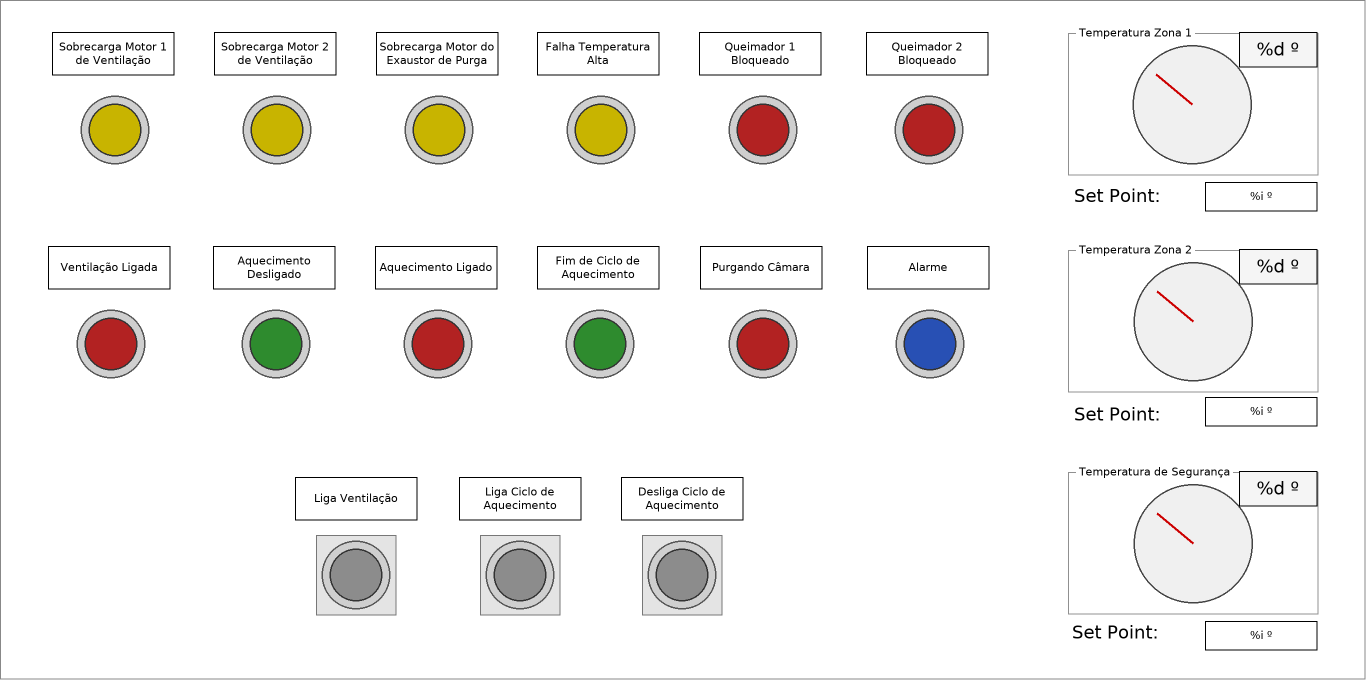
VISUALIZATION Manu021  // 1366x680
    Lamp1 (75,90 80x80), variable: GVL.sobrecarga_M1_vent_021, style: Lamp-Lamp1-Yellow
    Lamp1 (237,90 80x80), variable: GVL.sobrecarga_M2_vent_021, style: Lamp-Lamp1-Yellow
    Lamp1 (399,90 80x80), variable: GVL.sobrecarga_Purga_021, style: Lamp-Lamp1-Yellow
    Lamp1 (561,90 80x80), variable: GVL.falhaTempHigh_021, style: Lamp-Lamp1-Yellow
    Lamp1 (723,90 80x80), variable: GVL.queimador1_block_021, style: Lamp-Lamp1-Red
    Lamp1 (889,90 80x80), variable: GVL.queimador2_block_021, style: Lamp-Lamp1-Red
    Rectangle (52,32 122x43), "Sobrecarga Motor 1 de Ventilação"
    Rectangle (214,32 122x43), "Sobrecarga Motor 2 de Ventilação"
    Rectangle (376,32 122x43), "Sobrecarga Motor do Exaustor de Purga"
    Rectangle (537,32 122x43), "Falha Temperatura Alta"
    Rectangle (699,32 122x43), "Queimador 1 Bloqueado"
    Rectangle (866,32 122x43), "Queimador 2 Bloqueado"
    Lamp1 (71,304 80x80), variable: GVL.ventilacao_Ligada_021, style: Lamp-Lamp1-Red
    Rectangle (48,246 122x43), "Ventilação Ligada"
    Lamp1 (236,304 80x80), variable: GVL.aquecimento_Desligado_021, style: Lamp-Lamp1-Green
    Rectangle (213,246 122x43), "Aquecimento Desligado"
    Lamp1 (398,304 80x80), variable: GVL.aquecimento_Ligado_021, style: Lamp-Lamp1-Red
    Rectangle (375,246 122x43), "Aquecimento Ligado"
    Lamp1 (560,304 80x80), variable: GVL.fimCicloAquecimento_021, style: Lamp-Lamp1-Green
    Rectangle (537,246 122x43), "Fim de Ciclo de Aquecimento"
    Lamp1 (723,304 80x80), variable: GVL.purgandoCamara_021, style: Lamp-Lamp1-Red
    Rectangle (700,246 122x43), "Purgando Câmara"
    PushSwitch (316,535 80x80), variable: GVL.liga_ventilacao_021, behaviour: TAP, style: Switch-PushSwitch-Gray
    Rectangle (295,477 122x43), "Liga Ventilação"
    PushSwitch (480,535 80x80), variable: GVL.liga_aquecimento_021, behaviour: TAP, style: Switch-PushSwitch-Gray
    Rectangle (459,477 122x43), "Liga Ciclo de Aquecimento"
    PushSwitch (642,535 80x80), variable: GVL.desl_aquecimento_021, behaviour: TAP, style: Switch-PushSwitch-Gray
    Rectangle (621,477 122x43), "Desliga Ciclo de Aquecimento"
    Lamp1 (890,304 80x80), style: Lamp-Lamp1-Blue
    Rectangle (867,246 122x43), "Alarme"
    GroupBox (1068,25 250x150), "Temperatura Zona 1"
    Meter180 (1072,45 240x119), value: GVL.zona1atual_021, style: Meter-Meter180-Gray, scale format: %.1f, scale 20..160
        p518627256: ºC
    GroupBox (1068,242 250x150), "Temperatura Zona 2"
        Rectangle (171,7 78x35), "%d º", text variable: GVL.zona2atual_021
    Meter180 (1073,262 240x119), value: GVL.zona2atual_021, style: Meter-Meter180-Gray, scale format: %.1f, scale 20..160
        p518627256: ºC
    GroupBox (1068,464 250x150), "Temperatura de Segurança"
    Meter180 (1073,484 240x119), value: GVL.zonaSegAtual_021, style: Meter-Meter180-Gray, scale format: %.1f, scale 20..160
        p518627256: ºC
    Rectangle (1205,182 112x29), "%i º", text variable: GVL_P.zona1setpt_021
        OnMouseClick: write GVL_P.zona1setpt_021 via VisuDialogs.Numpad
    Label (1072,185 91x22), "Set Point:"
    Rectangle (1205,397 112x29), "%i º", text variable: GVL_P.zona2setpt_021
        OnMouseClick: write GVL_P.zona2setpt_021 via VisuDialogs.Numpad
    Label (1072,400 91x29), "Set Point:"
    Rectangle (1239,32 78x35), "%d º", text variable: GVL.zona1atual_021
    Rectangle (1239,471 78x35), "%d º", text variable: GVL.zonaSegAtual_021
    Label (1070,618 91x29), "Set Point:"
    Rectangle (1205,621 112x29), "%i º", text variable: GVL_P.zonaSegSetpt_021
        OnMouseClick: write GVL_P.zonaSegSetpt_021 via VisuDialogs.Numpad
END_VISUALIZATION

(* stored: Version 1.1.0.1, ProductVersion 3.1.4024.12
   Visu Manu021: Id {0ee97a16-888d-495f-ab73-8582710e6e5c} *)
